PROGRAM InfluxDb_WriteAlarms

VAR_INPUT
	IN_Dbid										: UINT;
	IN_FIFO										: FB_DBDatasetFifo_Influx;
	IN_Reset									: BOOL;
MesDataExd								: LoggerInfluxDb;
END_VAR

VAR
	// M_Init
		TP_Init									: TP;
		F_TRIG_Init								: F_TRIG;
   		bInit 									: BOOL;
	// Reset                					
		Trig_Reset								: R_TRIG;
	// Insert value             				
		CmdStart								: BOOL;
    	QueryOption_TSDB_Insert 				: T_QueryOptionTimeSeriesDB_Insert; // defines detailed Queryparameter
    	fbNoSQLQueryBuilder_TimeSeriesDB 		: FB_NoSQLQueryBuilder_TimeSeriesDB; // defines database type specific api
    	fbNoSqlQueryEvt 						: FB_NoSQLQueryEvt(sNetID := '', tTimeout := T#15S); // functionblock to execute queries
		nState 									: UINT;
		ValueToInsert							: ST_InfluxAlarmsInsert;
    // error handling helper values
    sErrorMessage								: STRING(255);

	
END_VAR

IF NOT bInit THEN
	M_Init();
END_IF

Trig_Reset(CLK := IN_Reset OR CmdClearFault_G);
IF Trig_Reset.Q THEN
	IN_Reset := FALSE;
	IN_FIFO.A_Reset();
END_IF

CmdStart := IN_FIFO.nCount >0 ;
IF CmdStart THEN
	CmdStart := FALSE;
	
	fbNoSQLQueryBuilder_TimeSeriesDB.pQueryOptions := ADR(QueryOption_TSDB_Insert);
	fbNoSQLQueryBuilder_TimeSeriesDB.cbQueryOptions := SIZEOF(QueryOption_TSDB_Insert);
	IN_FIFO.A_Get();
	ValueToInsert	:= IN_FIFO.Out;
	QueryOption_TSDB_Insert.sTableName 			:= 'Alarms';			
	QueryOption_TSDB_Insert.sDataType 			:= 'ST_InfluxAlarmsInsert';	
	QueryOption_TSDB_Insert.pSymbol 			:= ADR(ValueToInsert); 	
	QueryOption_TSDB_Insert.cbSymbol 			:= SIZEOF(ValueToInsert); 
	QueryOption_TSDB_Insert.nDataCount 			:= 1;					
	QueryOption_TSDB_Insert.nStartTimestamp 	:= F_GetSystemTime(); 	

	nState := 3;
END_IF

CASE nState OF 
    3:
        IF fbNoSqlQueryEvt.Execute(IN_Dbid, fbNoSQLQueryBuilder_TimeSeriesDB) THEN
			IF fbNoSqlQueryEvt.bError THEN
			MesDataExd.MesData.MesAlarmCode.1 := TRUE;
				nState := 1;
			ELSE
			MesDataExd.MesData.MesAlarmCode.1 := FALSE;
			   	nState := 1;
 				IN_FIFO.A_Remove();
           END_IF
        END_IF
END_CASE

METHOD M_Init : BOOL
VAR_INPUT
END_VAR
//Initialisation BUFFER
	//Buffer pour la lecture des sms
	IN_FIFO.A_Reset();
	IN_FIFO.A_Add();
	IN_FIFO.A_Get();
	IN_FIFO.A_Remove();
	
	IN_FIFO.In.Message :=  'Activation du code';
	IN_FIFO.A_Add();
	bInit := TRUE;
END_METHOD

END_PROGRAM

(* stored: Version 1.1.0.1, ProductVersion 3.1.4024.6
   POU InfluxDb_WriteAlarms: Id {e2894a4f-2143-4737-a5f6-066bb6aac3df}, SpecialFunc None
   Method M_Init: Id {a793e62f-35f2-46eb-bd07-7c32a8dd966b} *)
